FUNCTION_BLOCK BACnetAnalogOutput (* Service Interface Function Block Type *)
  (* Standard: 61499-2 *)
  (* Version 1.0, 2020-03-04, root *)
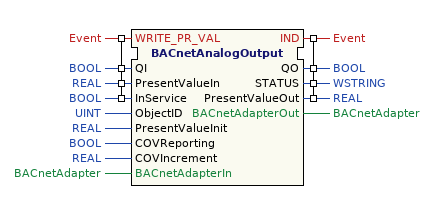
  EVENT_INPUT
    WRITE_PR_VAL WITH QI, PresentValueIn, InService; (* Service Initialization *)
  END_EVENT
  EVENT_OUTPUT
    IND WITH QO, STATUS, PresentValueOut; (* Indication from Resource *)
  END_EVENT
  VAR_INPUT
    QI : BOOL; (* Event Input Qualifier *)
    PresentValueIn : REAL;
    InService : BOOL;
    ObjectID : UINT;
    PresentValueInit : REAL;
    COVReporting : BOOL;
    COVIncrement : REAL;
  END_VAR
  VAR_OUTPUT
    QO : BOOL; (* Event Output Qualifier *)
    STATUS : WSTRING; (* Service Status *)
    PresentValueOut : REAL;
  END_VAR
  SOCKETS
    BACnetAdapterIn : BACnetAdapter;
  END_SOCKETS
  PLUGS
    BACnetAdapterOut : BACnetAdapter;
  END_PLUGS
END_FUNCTION_BLOCK
